{attribute 'qualified_only'}
{attribute 'strict'}
TYPE E_DOutputMode :
(
	AutoPLC 	:= 0,
	ManualHMI	:= 1
);
END_TYPE

(* stored: Version 1.1.0.1, ProductVersion 3.1.4024.12
   DUT E_DOutputMode: Id {e3ba8e88-e384-4ccd-9ff2-f8bbb7673404} *)
